// TIA Portal V19 export
TYPE "LAF_typePlasticWorkstationEm5ParametersInterface"
// stored: Access Published
   STRUCT
      configuration : "LAF_typePlasticWorkstationEm5Parameters";
      commands : "LBC_typeInterfaceCommands";
      monitoring { S7_SetPoint := 'True'} : "LAF_typePlasticWorkstationEm5ProcessValues";
   END_STRUCT;
END_TYPE
